(* Logix 5000 project; controller EuniceF_ICA17 vendor 1 type 14 code 150 rev 37.11; software revision 37.00 *)

TASK MainTask (continuous, watchdog 500 ms) : MainProgram

MODULES
   Local : vendor 1 type 14 code 150 (Compact 0, rev 37.11)
      Discrete_IO : Embedded (Compact 1, rev 3.1, Output RPI 20 ms)
      Analog_IO : Embedded (Compact 2, rev 1.1, Output RPI 80 ms)
      Counters : Embedded (Compact 3, rev 1.1, Output RPI 20 ms)
END_MODULES

VAR_GLOBAL   (* controller tags *)
   ALARM : BOOL;
   DoorOpen : BOOL;
   Keyswitch : BOOL;
   SEQ1 : DINT;
   SIREN : BOOL;
   Timer1 : TIMER := (PRE := 3000);
   Timer2 : TIMER := (PRE := 2000);
END_VAR

PROGRAM MainProgram   (* main routine MainRoutine *)

ROUTINE MainRoutine   (* ladder *)
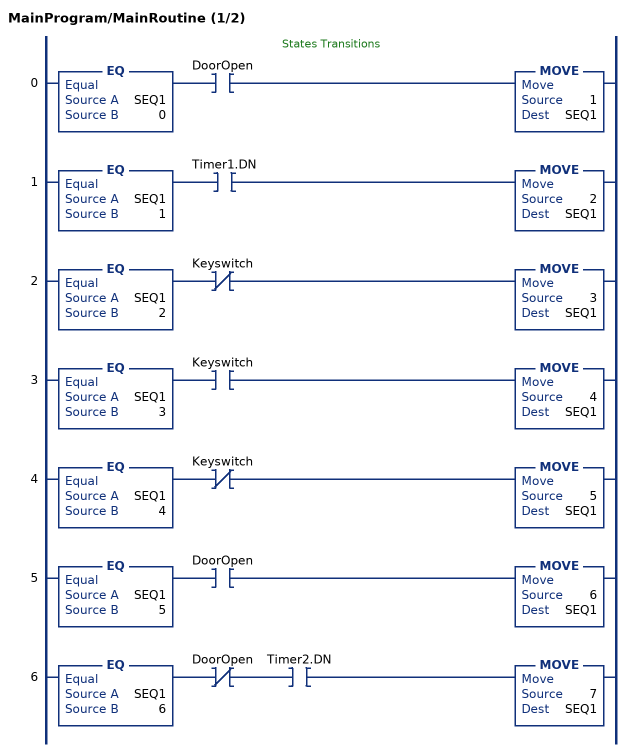
   // States Transitions
   0: EQ(SEQ1,0)XIC(DoorOpen)MOVE(1,SEQ1);
   1: EQ(SEQ1,1)XIC(Timer1.DN)MOVE(2,SEQ1);
   2: EQ(SEQ1,2)XIO(Keyswitch)MOVE(3,SEQ1);
   3: EQ(SEQ1,3)XIC(Keyswitch)MOVE(4,SEQ1);
   4: EQ(SEQ1,4)XIO(Keyswitch)MOVE(5,SEQ1);
   5: EQ(SEQ1,5)XIC(DoorOpen)MOVE(6,SEQ1);
   6: EQ(SEQ1,6)XIO(DoorOpen)XIC(Timer2.DN)MOVE(7,SEQ1);
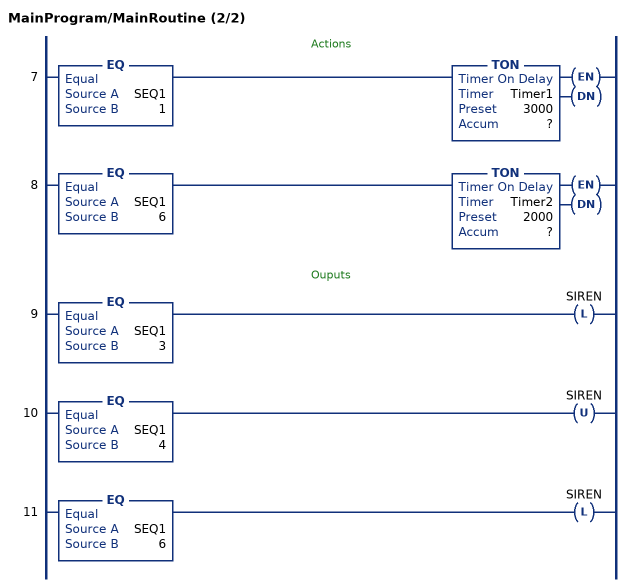
   // Actions
   7: EQ(SEQ1,1)TON(Timer1,?,?);
   8: EQ(SEQ1,6)TON(Timer2,?,?);
   // Ouputs
   9: EQ(SEQ1,3)OTL(SIREN);
   10: EQ(SEQ1,4)OTU(SIREN);
   11: EQ(SEQ1,6)OTL(SIREN);
END_ROUTINE
END_PROGRAM
